Omron CX-Programmer project NewProject (CX-Programmer 9.61)

# PLC TIMMER: CP1L M
; TES TIMMER

## Global symbols (name address type ; comment)
0.00 BOOL  ; START
0.01 BOOL  ; STOP
100.00 BOOL  ; K1
T0000 BOOL  ; TIMMER 00

## Program NewProgram1 (cyclic task 0)

### Section Section1

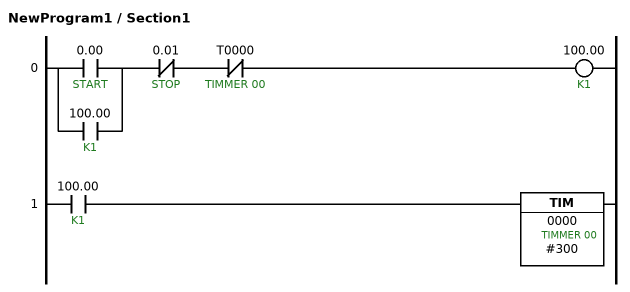
; rung 0
LD 0.00  ; START
OR 100.00  ; K1
ANDNOT 0.01  ; STOP
ANDNOT T0000  ; TIMMER 00
OUT 100.00  ; K1
; rung 1
LD 100.00  ; K1
TIM 0000 #300  ; TIMMER 00

### Section END
; rung 0
END(001)